Staubli VAL3: StopMotion.pgx

public program StopMotion()
begin
  //
  stopMove()
  taskKill("motion")
  wait(taskStatus("motion")==-1)
  resetMotion()
  call CloseSingnal()
  PublicData:libSave()
  popUpMsg("运动结束")
end
